Fanuc TP program (LS listing): RTR_TEST.LS

/PROG  RTR_TEST
/ATTR
OWNER		= MNEDITOR;
COMMENT		= "";
PROG_SIZE	= 1595;
CREATE		= DATE 22-03-26  TIME 07:20:28;
MODIFIED	= DATE 28-12-13  TIME 08:09:06;
FILE_NAME	= ;
VERSION		= 0;
LINE_COUNT	= 65;
MEMORY_SIZE	= 1971;
PROTECT		= READ_WRITE;
TCD:  STACK_SIZE	= 0,
      TASK_PRIORITY	= 50,
      TIME_SLICE	= 0,
      BUSY_LAMP_OFF	= 0,
      ABORT_REQUEST	= 0,
      PAUSE_REQUEST	= 0;
DEFAULT_GROUP	= 1,*,*,*,*;
CONTROL_CODE	= 00000000 00000000;
/APPL
/APPL

AUTO_SINGULARITY_HEADER;
  ENABLE_SINGULARITY_AVOIDANCE   : TRUE;
/MN
   1:   ;
   2:  CALL ROUTER(1) ;
   3:  CALL ROUTER(2) ;
   4:  CALL ROUTER(1) ;
   5:  CALL ROUTER(3) ;
   6:  CALL ROUTER(1) ;
   7:  CALL ROUTER(4) ;
   8:  CALL ROUTER(1) ;
   9:  CALL ROUTER(5) ;
  10:  CALL ROUTER(1) ;
  11:  CALL ROUTER(6) ;
  12:  CALL ROUTER(1) ;
  13:  CALL ROUTER(7) ;
  14:  CALL ROUTER(1) ;
  15:  CALL ROUTER(1) ;
  16:   ;
  17:  CALL ROUTER(2) ;
  18:  CALL ROUTER(3) ;
  19:  CALL ROUTER(2) ;
  20:  CALL ROUTER(4) ;
  21:  CALL ROUTER(2) ;
  22:  CALL ROUTER(5) ;
  23:  CALL ROUTER(2) ;
  24:  CALL ROUTER(6) ;
  25:  CALL ROUTER(2) ;
  26:  CALL ROUTER(7) ;
  27:  CALL ROUTER(2) ;
  28:  CALL ROUTER(2) ;
  29:   ;
  30:  CALL ROUTER(3) ;
  31:  CALL ROUTER(4) ;
  32:  CALL ROUTER(3) ;
  33:  CALL ROUTER(5) ;
  34:  CALL ROUTER(3) ;
  35:  CALL ROUTER(6) ;
  36:  CALL ROUTER(3) ;
  37:  CALL ROUTER(7) ;
  38:  CALL ROUTER(3) ;
  39:  CALL ROUTER(3) ;
  40:   ;
  41:  CALL ROUTER(4) ;
  42:  CALL ROUTER(5) ;
  43:  CALL ROUTER(4) ;
  44:  CALL ROUTER(6) ;
  45:  CALL ROUTER(4) ;
  46:  CALL ROUTER(7) ;
  47:  CALL ROUTER(4) ;
  48:  CALL ROUTER(4) ;
  49:   ;
  50:  CALL ROUTER(5) ;
  51:  CALL ROUTER(6) ;
  52:  CALL ROUTER(5) ;
  53:  CALL ROUTER(7) ;
  54:  CALL ROUTER(5) ;
  55:  CALL ROUTER(5) ;
  56:   ;
  57:  CALL ROUTER(6) ;
  58:  CALL ROUTER(7) ;
  59:  CALL ROUTER(6) ;
  60:  CALL ROUTER(6) ;
  61:   ;
  62:  CALL ROUTER(7) ;
  63:  CALL ROUTER(7) ;
  64:   ;
  65:  CALL ROUTER(1) ;
/POS
/END
